{attribute 'global_init_slot' := '40501'} 
TYPE ST_BaseElementIdentifier :
STRUCT
	stName					: ST_BaseLabel;
	sCode					: STRING;		//unikalny kod elementu w postaci X.X.X
	uiID					: UINT;			//unikalny numer elementu
	eType					: E_BaseElementType;
END_STRUCT
END_TYPE

(* stored: Version 1.1.0.1
   DUT ST_BaseElementIdentifier: Id {a640e5c6-59c4-4947-8e18-94accbba0643} *)
